# B&R Automation Studio project HMI
Automation Studio 4.8.2.72

## Configuration Config1

### Task classes (Cpu.sw)
```
Cyclic#4:
  Program <- Program.prg
VcDataObjects: Visu <- Visu.dob
```

### Hardware
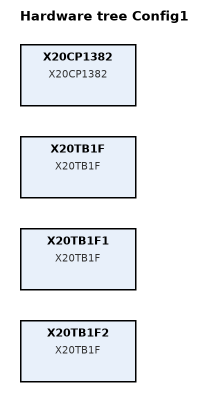
```
X20CP1382 : X20CP1382 v1.10.0.0  [X1 -> X1.SL; X2 -> X2.SL; X3 -> X3.SL]
  Module X1 (Type=X1, Virtual=true, Version=1.10.0.0)
    Connection (Connector=SS1, TargetModule=X20TB1F, TargetConnector=SS)
    Connection (Connector=SL, TargetModule=X20CP1382, TargetConnector=X1)
  Module X2 (Type=X2, Virtual=true, Version=1.10.0.0)
    Connection (Connector=SS1, TargetModule=X20TB1F1, TargetConnector=SS)
    Connection (Connector=SL, TargetModule=X20CP1382, TargetConnector=X2)
  Module X3 (Type=X3, Virtual=true, Version=1.10.0.0)
    Connection (Connector=SS1, TargetModule=X20TB1F2, TargetConnector=SS)
    Connection (Connector=SL, TargetModule=X20CP1382, TargetConnector=X3)
  Connector IF2:
    ActivateDevice = 1
    Mode = Manual
    InternetAddress = 127.0.0.1
    Vnc1
    VncVcObjectName1 = Visu
    VncKeyMappingFile1 = VC\PS2-Keyboard.dis
  ConfigurationID = HMI_Config1
  Simulation = 1
X20TB1F : X20TB1F v1.0.0.0
X20TB1F1 : X20TB1F v1.0.0.0
X20TB1F2 : X20TB1F v1.0.0.0
```

## Logical view

### Program Logical/Program (IEC)

#### Init.st - Init code
```iecst
PROGRAM _INIT
	(* Insert code here *)
	tmp := 20;

END_PROGRAM
```

#### Variables.var - Local variables
```iecst
VAR
	tmp : USINT;
END_VAR
```

- Visualisation Logical/Visu (not shown)

Listed in the project but not available here: Logical/Global.typ, Logical/Global.var, Logical/Libraries, Logical/Program/Cyclic.st, Logical/Program/Exit.st, Logical/Program/Types.typ
